// TIA Portal project "Proyecto2" (V16)

(* hardware
DEVICE "S7-1200 station_1"  S7-1200 Station
   slot 0: "Rack_0"  S7-1200 Rack  Rack  V1.0
   slot 1: "PLC_1"  CPU 1214C AC/DC/Rly  6ES7 214-1BG40-0XB0  V4.4
*)

// ===== PLC "PLC_1"  CPU 1214C AC/DC/Rly =====

VAR_GLOBAL   // PLC tag table "Tabla de variables estándar"
   ""pulsador"" AT %I0.0 : Bool;
   ""pulsador_start"" AT %I0.1 : Bool;
   ""pulsador_stop"" AT %I0.2 : Bool;
   ""motor"" AT %Q0.0 : Bool;
END_VAR